KUKA KRL program: sps_cycle_time.src, SPS_CYCLE_TIME.dat

--- sps_cycle_time.src ---
&ACCESS RV
&PARAM TEMPLATE = C:\KRC\Roboter\Template\ExpertVorgabe
&PARAM EDITMASK = *
DEFFCT REAL SPS_CYCLE_TIME(eProperty :IN)
DECL E_PROPERTY_CYCLE_TIME eProperty

IF VarState("eProperty") <> #INITIALIZED THEN
  eProperty = #GET
ENDIF

INT iTimernr
REAL rRet

SWITCH eProperty
CASE #SET
  iTimerNr = 20
  ; $TIMER[20], $TIMER_STOP[20]

  $TIMER_STOP[iTimerNr] = FALSE
  IF ($TIMER[iTimerNr] > 1000) OR ($TIMER[iTimerNr] < 0) THEN
     $TIMER[iTimerNr] = 0.0
  ENDIF

  rRet = $TIMER[iTimerNr]
  $TIMER[iTimerNr] = 0.0

  rCycleTime = rRet/1000
CASE #GET
  ;
ENDSWITCH

RETURN rCycleTime ; cycle time in seconds

END

--- SPS_CYCLE_TIME.dat ---
&ACCESS RV
&PARAM TEMPLATE = C:\KRC\Roboter\Template\ExpertVorgabe
&PARAM EDITMASK = *
DEFDAT SPS_CYCLE_TIME PUBLIC

GLOBAL ENUM E_PROPERTY_CYCLE_TIME GET, SET
REAL rCycleTime=0.0

ENDDAT
